VISUALIZATION VISU_State  // 12x17
VAR_IN_OUT
	state : BOOL;
	inactiveColor: Colors;
	activeColor : Colors;
END_VAR
    Ellipse (0,5 10x10), colour toggle: state, colour variable: inactiveColor
        p2167032090: activeColor
END_VISUALIZATION

(* stored: Version 1.1.0.1, ProductVersion 3.1.0.36
   Visu VISU_State: Id {89d064ec-c0a4-4d5b-90c2-a2d9a4e0e0e7} *)
